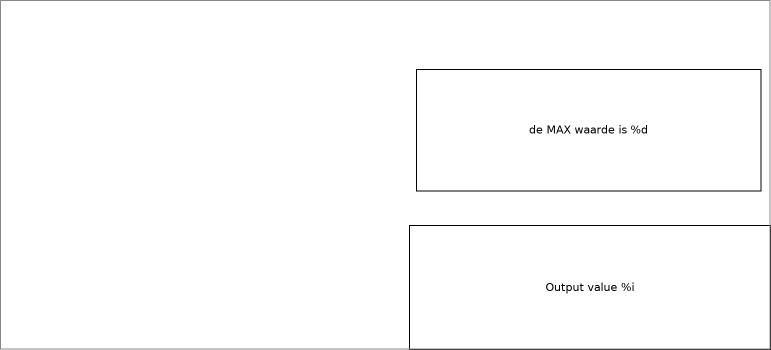
VISUALIZATION Visualization  // 771x350
    Rectangle (416,69 345x122), "de MAX waarde is %d", text variable: MAIN.NScale
        OnMouseClick: write the text variable via Default
    Rectangle (409,225 362x125), "Output value %i", text variable: MAIN.Apotentiometer
END_VISUALIZATION

(* stored: Version 1.1.0.1, ProductVersion 3.1.4024.12
   Visu Visualization: Id {693888ea-cbae-4b02-9db7-6a48c3bbad49} *)
